Fanuc KAREL source: kb00183.KL

PROGRAM KB00183
%NOLOCKGROUP
VAR
P1:INTEGER;P2:INTEGER;P3 : POSITION;P4:INTEGER
BEGIN
--
--
--
P1=1
P2=1
P4=1
SET_TRNS_TPE(P1,P2,P3,P4,1)
END KB00183
